FUNCTION_BLOCK trip_multiplexer (* Template for a simple Basic Function Block Type *)
  (* Standard: 61499-2 *)
  (* Version 1.0, 2021-02-26, badger *)
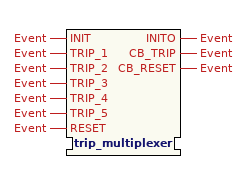
  EVENT_INPUT
    INIT; (* Initialization Request *)
    TRIP_1; (* Trip request 1 *)
    TRIP_2; (* Trip request 2 *)
    TRIP_3; (* Trip request 3 *)
    TRIP_4; (* Trip request 4 *)
    TRIP_5; (* Trip request 5 *)
    RESET; (* Reset the circuit breaker *)
  END_EVENT
  EVENT_OUTPUT
    INITO; (* Initialization Confirm *)
    CB_TRIP; (* Circuit Breaker output *)
    CB_RESET; (* Reset the circuit breaker *)
  END_EVENT
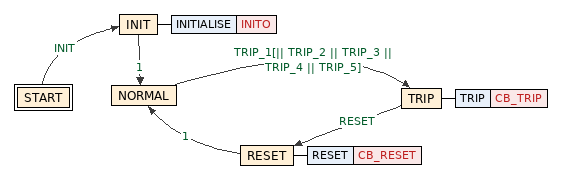
  EC_STATES
    START; (* Initial State *)
    INIT : INITIALISE -> INITO; (* Initialization *)
    TRIP : TRIP -> CB_TRIP; (* Normal execution *)
    NORMAL;
    RESET : RESET -> CB_RESET;
  END_STATES
  EC_TRANSITIONS
    START TO INIT := INIT;
    INIT TO NORMAL := 1;
    NORMAL TO TRIP := TRIP_1[|| TRIP_2  ||  TRIP_3 || TRIP_4 || TRIP_5]; (* Trigger if any of the trip request events are received. *)
    RESET TO NORMAL := 1;
    TRIP TO RESET := RESET; (* Reset the circuit breaker *)
  END_TRANSITIONS
  ALGORITHM INITIALISE IN AnyText: (* Initialization algorithm *)

  END_ALGORITHM
  ALGORITHM TRIP IN AnyText: (* Trip the circuit breaker *)

  END_ALGORITHM
  ALGORITHM RESET IN AnyText: (* Reset the circuit breaker *)

  END_ALGORITHM
END_FUNCTION_BLOCK
